FUNCTION_BLOCK TestType
  (* Version 0.1, 2005-04-08, Goran, Chalmers *)
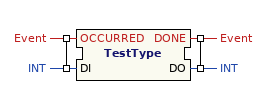
  EVENT_INPUT
    OCCURRED WITH DI;
  END_EVENT
  EVENT_OUTPUT
    DONE WITH DO;
  END_EVENT
  VAR_INPUT
    DI : INT;
  END_VAR
  VAR_OUTPUT
    DO : INT;
  END_VAR
  VAR
    invoked : INT;
  END_VAR
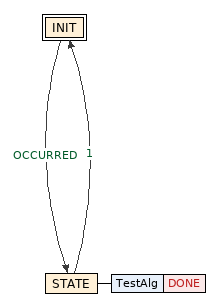
  EC_STATES
    INIT;
    STATE : TestAlg -> DONE;
  END_STATES
  EC_TRANSITIONS
    INIT TO STATE := OCCURRED;
    STATE TO INIT := 1;
  END_TRANSITIONS
  ALGORITHM TestAlg IN Java:
invoked = invoked + 1;
	DO = DI + 1;
	System.out.println("TestAlgorithm.execute():invoked: " + invoked + " times.");
	System.out.println("TestAlgorithm.execute(): DO: " + DO + ".");
  END_ALGORITHM
END_FUNCTION_BLOCK
